RoboDK station: QKM_robot_with_calibration_plate.rdk

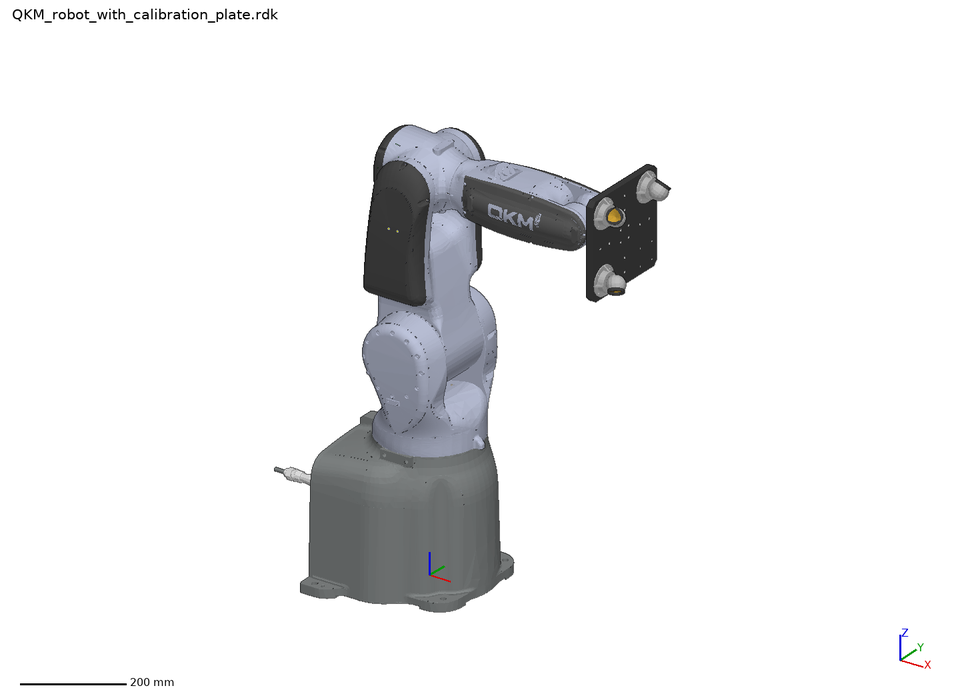
[picture v0: the station drawn from its stored meshes, robots at their saved joint values, targets as dots, program paths as lines]
Station QKM_robot_with_calibration_plate. Poses are relative to the parent item; angles as X-Y-Z fixed-axis rotations.
  - frame QKM HL6 Base at (0, 1000, 0) mm
    - robot QKM HL6: 6 axes
        modified DH rows (alpha deg, a mm, theta deg, d mm): 0, 0, 0, 491; -90, 0, -90, 0; 0, 350, -90, 0; -90, 0, 0, 350; 90, 0, 0, 0; -90, 0, 180, 84
        joint limits [-170, -110, -136, -185, -120, -360] to [170, 110, 136, 185, 120, 360]; home [0, 0, 90, 0, 0, 0]; saved at [0, 0, 90, 0, 0, 0]
      - tool , TCP at (0, 0, 15) mm, size 210 x 210 x 65.7 mm, geometry from 2.STEP
